// TIA Portal V20 export
DATA_BLOCK "CMInterface_Filling_DB"   // DB82
// stored: InstanceOfName CM_Interface_Filling, InstanceOfType FB
"CM_Interface_Filling"
   // VAR_INPUT
   //    CmCommand { ExternalAccessible := 'False'; ExternalVisible := 'False'; ExternalWritable := 'False'} : Array[0..29] of Bool;
   //    Procedure_Param { ExternalAccessible := 'False'; ExternalVisible := 'False'; ExternalWritable := 'False'} : Array[0..31] of Real;
   //    ProcessValue_In : Array[0..31] of Real;
   //    CmFbOnOff { ExternalAccessible := 'False'; ExternalVisible := 'False'; ExternalWritable := 'False'} : Array[0..29] of Bool;
   //    Auto_Man : Bool;
   //    Oos : Bool;
   // END_VAR
   // VAR_OUTPUT
   //    CM_V101 { ExternalAccessible := 'False'; ExternalVisible := 'False'; ExternalWritable := 'False'} : "DigVal";
   //    CM_V100 { ExternalAccessible := 'False'; ExternalVisible := 'False'; ExternalWritable := 'False'} : "DigVal";
   //    FillingSpeedSilo1 : "AnaVal";
   //    FillingSpeedSilo2 : "AnaVal";
   //    FillingSpeedSilo3 : "AnaVal";
   //    FillingSpeedCleaning : "AnaVal";
   //    FillingSpeedAllSilo : "AnaVal";
   // END_VAR
   // VAR
   //    Pos_edge : Bool;
   //    Neg_edge : Bool;
   // END_VAR
BEGIN
END_DATA_BLOCK
